Staubli VAL3: WriteSingleIO.dtx

public bool bState
public num nModuleId
public num nPin
